(* CODESYS project Bronkhorst.library
   Author: Ziga Javornik
   Version: 0.0.3.1
   Description: Various bronkhorst device impleentations.
   Title: ZigaLibs.Bronkhorst
   Placeholder: ZigaLibs.Bronkhorst
   DefaultNamespace: ZigaLibs.Bronkhorst
   Company: Ziga Javornik

Project tree, tasks and I/O mapping:
  libraries: Tc2_Standard, * (Beckhoff Automation GmbH); Tc2_System, * (Beckhoff Automation GmbH); Tc3_Module, * (Beckhoff Automation GmbH); TcUnit, 1.3.1 (www.tcunit.org); ZigaLibs.Core, 0.0.3.7 (Ziga Javornik); ZigaLibs.Logging, 0.0.4.1 (Ziga Javornik)
  GVLs/
  SOURCE/
    MassFlow or PressureController/
      DUTs/
        data type E_ControllerMode
        data type E_ParameterReadingStep
        data type ST_ControllerCoeList
        data type ST_ControllerInputs
        data type ST_ControllerOutputs
        data type ST_ControllerStatus
      POUs/
        function block FB_FlowController [ST]: FB_init, CalculateMeasuredValue, CalculateSetpointValue, ControllerModeWriting, ControllerSpeedWriting, ReadCoE, Capacity, CapacityUnit, ControllerSpeed, FluidName, Mode, Status
    program FlowUnits [ST]: Bar, LsMin, Sccm, Slm
    program GasTypes [ST]: Air, BBr3, BCl3, C2F6, Cl2, H2, He, N2, O2, SF6, SiF4
  TESTS/
    Test suites/
      function block FB_FlowController_Tests [ST]: Test01_MeasuredValueConversion_1000, Test02_MeasuredValueConversion_32767, Test03_MeasuredValueConversion_0, Test04_MeassuredValueConversion_decimalDigits0, Test05_SetpointValueConversion_1000, Test06_SetpointValueConversion_10000, Test07_SetpointValueConversion_0, Test08_SetpointValueConversion_decimalDigits0, Test09_EnablePreventsOutoutFlowAndSetsControlByteToZero, Test10_ControllerStatusConversion, Test11_ValvePosition
      function block FB_FlowUnits_Tests [ST]: Test_AllFlowUnits
      function block FB_GasTypes_Tests [ST]: Test_AllGasTypes
    program PRG_TESTS [ST]
*)

// SOURCE/MassFlow or PressureController/DUTs/E_ControllerMode
{attribute 'qualified_only'}
{attribute 'to_string'}
TYPE E_ControllerMode :
(
	Controlling 	:= 16#80,	// Control at setpoint value
	ValveClosed		:= 16#83,	// No controller action, valve is closed
	ControllerIdle	:= 16#84,	// No controller action, valve remains its position 
	ValvePurge		:= 16#88	// No controller action, valve is fully open
)USINT;
END_TYPE

// SOURCE/MassFlow or PressureController/DUTs/E_ParameterReadingStep
{attribute 'qualified_only'}
{attribute 'strict'}
TYPE E_ParameterReadingStep :
(
	IDLE,
	GAS_TYPE,
	FLOW_UNIT,
	DECIMAL_DIGITS,
	FLOW_CAPACITY
);
END_TYPE

// SOURCE/MassFlow or PressureController/DUTs/ST_ControllerCoeList
// Contains CoE indexes and sub indexes for Bronkhorst EtherCAT mass flow controller
TYPE ST_ControllerCoeList :
STRUCT
	FluidName		: ZigaLibs_Core.ST_CoeEntry_String30 	:= (Index := 16#2001, SubIndex := 16#12);
	Capacity 		: ZigaLibs_Core.ST_CoeEntry_REAL 		:= (Index := 16#2001, SubIndex := 16#0E);
	CapacityUnit 	: ZigaLibs_Core.ST_CoeEntry_String30 	:= (Index := 16#2001, SubIndex := 16#20);
	DecimalDigits 	: ZigaLibs_Core.ST_CoeEntry_INT 		:= (Index := 16#6407, SubIndex := 16#01);
	ControlMode 	: ZigaLibs_Core.ST_CoeEntry_USINT 		:= (Index := 16#6423, SubIndex := 16#01);
	ControllerSpeed	: ZigaLibs_Core.ST_CoeEntry_USINT		:= (Index := 16#2072, Subindex := 16#1F);
END_STRUCT
END_TYPE

// SOURCE/MassFlow or PressureController/DUTs/ST_ControllerInputs
TYPE ST_ControllerInputs :
STRUCT
	MeassuredValue	: INT;
	ValvePosition	: UINT;
	StatusWord		: UINT;
	AmsAddr			: Tc2_System.ST_AmsAddr;
END_STRUCT
END_TYPE

// SOURCE/MassFlow or PressureController/DUTs/ST_ControllerOutputs
TYPE ST_ControllerOutputs :
STRUCT
	ControlByte	: USINT;
	Setpoint	: INT;
END_STRUCT
END_TYPE

// SOURCE/MassFlow or PressureController/DUTs/ST_ControllerStatus

TYPE ST_ControllerStatus :
STRUCT
	ControllerOn		: BOOL;
	SelfOptimization	: BOOL;
	ManualMode			: BOOL;
	SetpointSwitch		: BOOL;
	OptimizationError	: BOOL;
	DataNotValid		: BOOL;
	Overload			: BOOL;
	NetOverload			: BOOL;
END_STRUCT
END_TYPE

// SOURCE/MassFlow or PressureController/POUs/FB_FlowController
(* Bronkhorst mass flow/pressure controller device implementation.
============================================================================================================================================================================================
CONSTRUCTOR TEMPLATE - COPY EVERYTHING BELOW, ADJUST PARAMETERS ACCORDINGLY!
============================================================================================================================================================================================	
(fPredictedFlowCapacity	:= 100, // [REAL] Predicted flow capacity. If logger is provided and the read capacity differs, the error will be reported by the logger.
sPredictedGasType := N2, // [STRING] Predicted gas type. If logger is provided and the read gas type differs, the error will be reported by the logger.
sPredictedFlowUnit := sccm, // [STRING] Predicted flow unit. If logger is provided and the read flow unit differs, the error will be reported by the logger.
iLogger := 0, // [ZigaLibs_Core.I_LoggerEx] Logger implementation provided, set to 0 if not required.
mode := E_ControllerMode.Controlling); // [E_ControllerMode] Controller initial mode
============================================================================================================================================================================================
*)

FUNCTION_BLOCK FB_FlowController EXTENDS ZigaLibs_Core.FB_HasInstanceNameAndPath
VAR_INPUT
	bEnable				: BOOL;	// Enables controller
	fSetpoint			: REAL;	// Setpoint to the controller
	bReadParameters		: BOOL; // Reads CoE parameters on rising edge trigger
END_VAR
VAR_OUTPUT
	fMeassuredValue	: REAL;	// Measured value, reported from the controller
	fValvePosition	: REAL;	// Valve position
END_VAR

// IO
VAR
	Inputs	AT %I*	: ST_ControllerInputs;
	Outputs	AT %Q* 	: ST_ControllerOutputs;
END_VAR

VAR
	bFirstExecution			: BOOL := TRUE;
	_stringBuilder			: ZigaLibs_Core.FB_StringBuilder;
	_CoeList				: ST_ControllerCoeList;
	_logPrefix				: STRING := Tc2_Standard.CONCAT(STR1 := _instancePath, STR2 := ': ');
	_logger					: REFERENCE TO ZigaLibs_Logging.I_Logger;
	_writeLogs				: BOOL;
	_ethercatBoxName		: Tc2_System.T_MaxString;
	{attribute 'hide'} 
	_mode					: E_ControllerMode;	// Hide since mode switching should be logged (done inside the property setter)
	_status					: ST_ControllerStatus;
	_predictedFlowCapacity	: REAL;
	_predictedGasType		: STRING;
	_predictedFlowUnit		: STRING;
	_writeModeRequired					: BOOL;
	_validateModeWrite					: BOOL;
	_controlModeTmp						: E_ControllerMode;
	_coeReadWrite						: ZigaLibs_Core.FB_CoeReadWrite;
	_readParametersRequest				: Tc2_Standard.R_TRIG;
	_parametersReadingInProgress		: BOOL;
	_readBoxName						: ZigaLibs_Core.FB_ReadBoxName;
	_controllerSpeed					: UINT := 1;
	_updateControllerSpeedRequired		: BOOL;
	_validateControllerSpeed			: BOOL;
END_VAR

VAR CONSTANT
	VALVE_FULLY_OPENED_VALUE : REAL := 617.0;
END_VAR

Outputs.ControlByte := BOOL_TO_BYTE(bEnable);

IF bEnable THEN
	Outputs.Setpoint := CalculateSetpointValue();
ELSE
	Outputs.Setpoint := 0;
END_IF

fMeassuredValue := CalculateMeasuredValue();
fValvePosition := 100.0 * UINT_TO_REAL(Inputs.ValvePosition)/VALVE_FULLY_OPENED_VALUE;

IF bFirstExecution THEN
	IF ReadCoE() THEN
		bFirstExecution := FALSE;
	END_IF
END_IF

_readParametersRequest(CLK := bReadParameters);
// Parameters read request
IF _readParametersRequest.Q THEN
	_parametersReadingInProgress := TRUE;
END_IF

IF _parametersReadingInProgress THEN
	IF ReadCoE() THEN
		_parametersReadingInProgress := FALSE;
	END_IF
END_IF

// Controller mode writing and validation
ControllerModeWriting();
// Controller speed writing and validation
ControllerSpeedWriting();

// Status of the controller
_status.ControllerOn := Inputs.StatusWord.0;
_status.SelfOptimization := Inputs.StatusWord.1;
_status.ManualMode := Inputs.StatusWord.2;
_status.SetpointSwitch := Inputs.StatusWord.3;
_status.OptimizationError := Inputs.StatusWord.4;
_status.DataNotValid := Inputs.StatusWord.8;
_status.Overload := Inputs.StatusWord.9;
_status.NetOverload := Inputs.StatusWord.10;

METHOD FB_init : BOOL
VAR_INPUT
	bInitRetains : BOOL; // if TRUE, the retain variables are initialized (warm start / cold start)
	bInCopyCode : BOOL;  // if TRUE, the instance afterwards gets moved into the copy code (online change)
	
	fPredictedFlowCapacity	: REAL;	// Predicted flow capacity. If bWriteLogs is set to TRUE and the read capacity differs, the error will be reported by the logger.
	sPredictedGasType		: STRING;// Predicted gas type. If bWriteLogs is set to TRUE and the read gas type differs, the error will be reported by the logger.
	sPredictedFlowUnit		: STRING; // Predicted flow unit. If bWriteLogs is set to TRUE and the read flow unit differs, the error will be reported by the logger.
	logger					: REFERENCE TO ZigaLibs_Logging.I_Logger;	// Logger implementation provided, set to 0 if not required.
	mode					: E_ControllerMode;	// Controller initial mode
END_VAR
_predictedFlowCapacity := fPredictedFlowCapacity;
_predictedGasType := sPredictedGasType;
_predictedFlowUnit := sPredictedFlowUnit;
_logger REF= logger;
_mode := mode;
_writeLogs := __ISVALIDREF(logger);
END_METHOD

METHOD PRIVATE CalculateMeasuredValue : REAL
VAR_INPUT
END_VAR
CalculateMeasuredValue :=  INT_TO_REAL(Inputs.MeassuredValue) / LREAL_TO_REAL(EXPT(10,_CoeList.DecimalDigits.Value));
END_METHOD

METHOD PRIVATE CalculateSetpointValue : INT
VAR_INPUT
END_VAR
CalculateSetpointValue := REAL_TO_INT(fSetpoint * LREAL_TO_REAL(EXPT(10, _CoeList.DecimalDigits.Value)));
END_METHOD

METHOD PRIVATE ControllerModeWriting
IF _writeModeRequired AND_THEN _coeReadWrite.WriteAny(
		CoeEntry := ADR(_CoeList.ControlMode),
		Value := _mode,
		SlaveAddr := Inputs.AmsAddr)
THEN
	IF _writeLogs THEN
		_logger.LogInfo(message := _stringBuilder.Reset()
			.AddString(str := _logPrefix)
			.AddString(str := 'Finished writing control mode for EtherCAT device ')
			.AddWithDblQuotationMarks(str := _ethercatBoxName)
			.AddString(str := '.')
			.Create());
	END_IF
	_validateModeWrite := TRUE;
	_writeModeRequired := FALSE;
END_IF

IF _validateModeWrite AND_THEN _coeReadWrite.ReadAny(
		CoeEntry := ADR(_CoeList.ControlMode),
		Value := _CoeList.ControlMode.Value,
		SlaveAddr := Inputs.AmsAddr)
THEN
	_validateModeWrite := FALSE;
	IF _writeLogs THEN
		IF _CoeList.ControlMode.Value <> _mode THEN
			// This allows for using TO_STRING on the enum value for better logging experience.
			_controlModeTmp := _CoeList.ControlMode.Value;
			_logger.LogError(message := _stringBuilder.Reset()
				.AddString(str := _logPRefix)
				.AddString('Control mode validation failed! Actual mode read is ')
				.AddWithDblQuotationMarks(str := TO_STRING(_controlModeTmp))
				.AddString(' required mode is ')
				.AddWithDblQuotationMarks(str := TO_STRING(_mode))
				.Create());
		ELSE
			_logger.LogInfo(message := _stringBuilder.Reset()
				.AddString(str := _logPrefix)
				.AddString('Control mode setting validation successful.')
				.Create());
		END_IF
	END_IF
END_IF
END_METHOD

METHOD PRIVATE ControllerSpeedWriting
VAR_INPUT
END_VAR
IF _updateControllerSpeedRequired AND_THEN _coeReadWrite.WriteAny(
		CoeEntry := ADR(_CoeList.ControllerSpeed),
		Value := _controllerSpeed,
		SlaveAddr := Inputs.AmsAddr)
THEN
	IF _writeLogs THEN
	_logger.LogInfo(message := _stringBuilder.Reset()
		.AddString(str := _logPrefix)
		.AddString(str := 'Finished writing controller speed for EtherCAT device ')
		.AddWithDblQuotationMarks(str := _ethercatBoxName)
		.AddString(str := '.')
		.Create());
	END_IF
	_validateControllerSpeed := TRUE;
	_updateControllerSpeedRequired := FALSE;
END_IF

IF _validateControllerSpeed AND_THEN _coeReadWrite.ReadAny(
		CoeEntry := ADR(_CoeList.ControllerSpeed),
		Value := _CoeList.ControlMode.Value,
		SlaveAddr := Inputs.AmsAddr)
THEN
	_validateControllerSpeed := FALSE;
	IF _writeLogs THEN
		IF _CoeList.ControlMode.Value <> _mode THEN
			_logger.LogError(message := _stringBuilder.Reset()
				.AddString(str := _logPRefix)
				.AddString('Control speed validation failed! Actual speed read is ')
				.AddWithDblQuotationMarks(str := TO_STRING(_CoeList.ControllerSpeed.Value))
				.AddString(' required speed is ')
				.AddWithDblQuotationMarks(str := TO_STRING(_controllerSpeed))
				.Create());
		ELSE
			_logger.LogInfo(message := _stringBuilder.Reset()
				.AddString(str := _logPrefix)
				.AddString('Control speed setting validation successful.')
				.Create());
		END_IF
	END_IF
END_IF
END_METHOD

(* Reads CoE items and updates them. Returns TRUE when done, even if an error occurs. Error is reported to log.*)
METHOD PRIVATE ReadCoE : BOOL
VAR_INST
	eReadCoeStep	: E_ParameterReadingStep;
	bCoeReadError	: BOOL;
	bError			: BOOL;
	fbCoeReadWrite	: ZigaLibs_Core.FB_CoeReadWrite;
END_VAR

VAR CONSTANT
	MAX_REAL_VALUE_DEVIATION : REAL := 0.1;
END_VAR

VAR_INST
	message	: Tc2_System.T_MaxString;
	mfcName	: Tc2_System.T_MaxString;
END_VAR
CASE eReadCoeStep OF
	E_ParameterReadingStep.IDLE:
		ReadCoE := FALSE;
		message := '';
		IF _ethercatBoxName = '' THEN
			_readBoxName(
				AmsNetId := Inputs.AmsAddr,
				PlcRuntimeNetId := '',
				error => bError,
				name => _ethercatBoxName);
		ELSIF _ethercatBoxName <> '' OR bError THEN
			eReadCoeStep := E_ParameterReadingStep.GAS_TYPE;
			IF _writeLogs THEN
				IF NOT bError THEN
					message := _stringBuilder.Reset()	
						.AddString(str := _logPrefix)
						.AddString(str := 'MFC parameters ')
						.AddWithDblQuotationMarks(str := _ethercatBoxName)
						.AddString(str := ':')
						.Create();
				ELSE
					_logger.LogInfo(message := _stringBuilder.Reset()	
						.AddString(str := _logPrefix)
						.AddString(str := 'Reading CoE parameters for Bronkhorst device ')
						.AddWithDblQuotationMarks(str := '<Error reading EC box name>')
						.AddString(str := '...')
						.Create());
				END_IF

			END_IF
		END_IF
		
	E_ParameterReadingStep.GAS_TYPE:
		IF fbCoeReadWrite.ReadAny(
			CoeEntry := ADR(_CoeList.FluidName),
			Value := _CoeList.FluidName.Value,
			SlaveAddr := Inputs.AmsAddr)
		THEN
			_CoeList.FluidName.Value := ZigaLibs_Core.StringHelper.TrimRightSide(_CoeList.FluidName.Value);
			IF _writeLogs THEN
				IF ZigaLibs_Core.StringHelper.TrimRightSide(_CoeList.FluidName.Value) <> _predictedGasType THEN
					_logger.LogWarning(message := _stringBuilder.Reset()
						.AddString(_logPrefix)
						.AddString('Invalid gas type found! Predicted gas type is ')
						.AddWithDblQuotationMarks(_predictedGasType)
						.AddString(' and actual gas type found is ')
						.AddWithDblQuotationMarks(_coeList.FluidName.Value)
						.Create());
				ELSE
					message :=_stringBuilder.Reset()
						.AddString(message)
						.AddString('[')
						.AddString('Gas type: ')
						.AddWithDblQuotationMarks(_coeList.FluidName.Value)
						.AddString(']')
						.Create();
				END_IF
			END_IF
			eReadCoeStep := E_ParameterReadingStep.FLOW_UNIT;
		END_IF
		
	E_ParameterReadingStep.FLOW_UNIT:
		IF fbCoeReadWrite.ReadAny(
			CoeEntry := ADR(_CoeList.CapacityUnit),
			Value := _CoeList.CapacityUnit.Value,
			SlaveAddr := Inputs.AmsAddr)
		THEN
			_CoeList.CapacityUnit.Value := ZigaLibs_Core.StringHelper.TrimRightSide(_CoeList.CapacityUnit.Value);
			IF _writeLogs THEN
				IF ZigaLibs_Core.StringHelper.TrimRightSide(_CoeList.CapacityUnit.Value) <> _predictedFlowUnit THEN
					_logger.LogWarning(message := _stringBuilder.Reset()
						.AddString(_logPrefix)
						.AddString('Invalid flow unit found! Predicted unit is ')
						.AddWithDblQuotationMarks(_predictedFlowUnit)
						.AddString(' and actual flow unit found is ')
						.AddWithDblQuotationMarks(_coeList.CapacityUnit.Value)
						.Create());				
				ELSE
					message :=_stringBuilder.Reset()
						.AddString(message)
						.AddString('[')
						.AddString('Flow unit: ')
						.AddWithDblQuotationMarks(_coeList.CapacityUnit.Value)
						.AddString(']')
						.Create();
				END_IF
			END_IF
			eReadCoeStep := E_ParameterReadingStep.DECIMAL_DIGITS;
		END_IF
		
	E_ParameterReadingStep.DECIMAL_DIGITS:
		IF fbCoeReadWrite.ReadAny(
			CoeEntry := ADR(_CoeList.DecimalDigits),
			Value := _CoeList.DecimalDigits.Value,
			SlaveAddr := Inputs.AmsAddr)
		THEN
			eReadCoeStep := E_ParameterReadingStep.FLOW_CAPACITY;
		END_IF
		
	E_ParameterReadingStep.FLOW_CAPACITY:
		IF fbCoeReadWrite.ReadAny(
			CoeEntry := ADR(_CoeList.Capacity),
			Value := _CoeList.Capacity.Value,
			SlaveAddr := Inputs.AmsAddr)
		THEN
			IF _writeLogs THEN
				IF ABS(_CoeList.Capacity.Value - _predictedFlowCapacity) >= MAX_REAL_VALUE_DEVIATION THEN
					_logger.LogWarning(message := _stringBuilder.Reset()
						.AddString(_logPrefix)
						.AddString('Invalid flow capacity found! Predicted capacity is ')
						.AddString(ZigaLibs_Core.StringConstants.DoubleQuotationMark)
						.AddAnyReal(_predictedFlowCapacity, 3, TRUE).AddString(' ').AddString(_coeList.CapacityUnit.Value)
						.AddString(ZigaLibs_Core.StringConstants.DoubleQuotationMark)
						.AddString(' and actual flow capacity found is ')
						.AddString(ZigaLibs_Core.StringConstants.DoubleQuotationMark)
						.AddAnyReal(_CoeList.Capacity.Value, 3, TRUE).AddString(' ').AddString(_coeList.CapacityUnit.Value)
						.AddString(ZigaLibs_Core.StringConstants.DoubleQuotationMark)
						.AddString('!')
						.Create());
					ELSE
							
					message :=_stringBuilder.Reset()
						.AddString(message)
						.AddString('[')
						.AddString('Flow capacity: ')
						.AddString(ZigaLibs_Core.StringConstants.DoubleQuotationMark)
						.AddAnyReal(_CoeList.Capacity.Value, 3, TRUE).AddString(' ').AddString(_coeList.CapacityUnit.Value)
						.AddString(ZigaLibs_Core.StringConstants.DoubleQuotationMark)
						.AddString(']')
						.Create();
						
					_logger.LogInfo(message);
					END_IF
				END_IF
			eReadCoeStep := E_ParameterReadingStep.IDLE;
			ReadCoE := TRUE;
		END_IF	
END_CASE
END_METHOD

{attribute 'monitoring':='call'}
// Gets capacity of the device
PROPERTY Capacity : REAL
GET
Capacity := _CoeList.Capacity.Value;
END_GET
END_PROPERTY

{attribute 'monitoring':='call'}
// Gets the capacity unit of the device
PROPERTY CapacityUnit : STRING(30)
GET
CapacityUnit := _CoeList.CapacityUnit.Value;
END_GET
END_PROPERTY

{attribute 'monitoring'='call'}
(*Gets or sets the controller speed.
The controller speed is default set on 1, increasing THIS number will make it faster. 
Please be aware that increasing the controller speed can lead to oscillation when setpoint steps are to steep, 
this will need to be fine-tuned on site to find the optimum setting for the process*)
PROPERTY PUBLIC ControllerSpeed : UINT := 1
GET
ControllerSpeed := _controllerSpeed;
END_GET
SET
IF ControllerSpeed <> _controllerSpeed THEN
	_updateControllerSpeedRequired := TRUE;
END_IF
_controllerSpeed := ControllerSpeed;
END_SET
END_PROPERTY

{attribute 'monitoring':='call'}
// Gets the fluid name of the device
PROPERTY FluidName : STRING(30)
GET
FluidName := _CoeList.FluidName.Value;
END_GET
END_PROPERTY

{attribute 'monitoring':='call'}
// Gets or sets the controller mode
PROPERTY PUBLIC Mode : E_ControllerMode
GET
Mode := _mode;
END_GET
SET
IF _mode <> Mode THEN
	_writeModeRequired := TRUE;
END_IF

_mode := Mode;
END_SET
END_PROPERTY

{attribute 'monitoring':='call'}
// Gets the controller status
PROPERTY Status : REFERENCE TO ST_ControllerStatus
GET
Status REF= _status;
END_GET
END_PROPERTY

END_FUNCTION_BLOCK

// SOURCE/FlowUnits
PROGRAM FlowUnits
VAR
END_VAR

PROPERTY Bar : string
GET
Bar := 'bar(g)';
END_GET
END_PROPERTY

PROPERTY PUBLIC LsMin : STRING
GET
LsMin := 'ls/min';
END_GET
END_PROPERTY

PROPERTY Sccm : STRING
GET
Sccm := 'sccm';
END_GET
END_PROPERTY

PROPERTY Slm : STRING
GET
Slm := 'slm';
END_GET
END_PROPERTY

END_PROGRAM

// SOURCE/GasTypes
{attribute 'no_explicit_call' := 'Body contains no logic, calling methods only allowed.'}
{attribute 'hide_all_locals'}

// A class containing possible gas types for Bronkhorst devices stored as a string.
PROGRAM GasTypes
VAR
END_VAR

{attribute 'monitoring':='call}
PROPERTY Air : STRING
GET
Air := 'AiR';
END_GET
END_PROPERTY

{attribute 'monitoring':='variable'}
PROPERTY BBr3 : STRING
GET
BBr3 := 'BBr3';
END_GET
END_PROPERTY

{attribute 'monitoring':='variable'}
PROPERTY BCl3 : STRING
GET
BCl3 := 'BCl3';
END_GET
END_PROPERTY

{attribute 'monitoring':='variable'}
PROPERTY C2F6 : STRING
GET
C2F6 := 'C2F6';
END_GET
END_PROPERTY

{attribute 'monitoring':='variable'}
PROPERTY Cl2 : STRING
GET
Cl2 := 'Cl2';
END_GET
END_PROPERTY

{attribute 'monitoring':='variable'}
PROPERTY H2 : STRING
GET
H2 := 'H2';
END_GET
END_PROPERTY

{attribute 'monitoring':='variable'}
PROPERTY He : STRING
GET
He := 'He';
END_GET
END_PROPERTY

{attribute 'monitoring':='variable'}
PROPERTY N2 : STRING
GET
N2 := 'N2';
END_GET
END_PROPERTY

{attribute 'monitoring':='variable'}
PROPERTY O2 : STRING
GET
O2 := 'O2';
END_GET
END_PROPERTY

{attribute 'monitoring':='variable'}
PROPERTY SF6 : STRING
GET
SF6 := 'SF6';
END_GET
END_PROPERTY

{attribute 'monitoring':='variable'}
PROPERTY SiF4 : STRING
GET
SiF4 := 'SiF4';
END_GET
END_PROPERTY

END_PROGRAM

// TESTS/Test suites/FB_FlowController_Tests
// Subject under test
FUNCTION_BLOCK INTERNAL FB_FlowController_Tests EXTENDS TcUnit.FB_TestSuite

// Create instance variables that will be accesible for all tests
VAR
	_mfc : FB_FlowController(	
		fPredictedFlowCapacity	:= 0.0,	// Predicted flow capacity. If bLogInvalidParams is set to TRUE and the read capacity differs, the error will be reported by the logger.
		sPredictedGasType		:= 'Cl2',// Predicted gas type. If bLogInvalidParams is set to TRUE and the read gas type differs, the error will be reported by the logger.
		sPredictedFlowUnit		:= 'sccm', // Predicted flow unit. If bLogInvalidParams is set to TRUE and the read flow unit differs, the error will be reported by the logger.
		logger					:= 0,	// Logger implementation provided
		mode					:= E_ControllerMode.Controlling);
END_VAR

// Call your test methods here
Test01_MeasuredValueConversion_1000();
Test02_MeasuredValueConversion_32767();
Test03_MeasuredValueConversion_0();
Test04_MeassuredValueConversion_decimalDigits0();
Test05_SetpointValueConversion_1000();
Test06_SetpointValueConversion_10000();
Test07_SetpointValueConversion_0();
Test08_SetpointValueConversion_decimalDigits0();
Test09_EnablePreventsOutoutFlowAndSetsControlByteToZero();
Test10_ControllerStatusConversion();
Test11_ValvePosition();

METHOD PRIVATE Test01_MeasuredValueConversion_1000

(* Instanced variables are VERY useful for writing tests since tests are run in paralel (by default).
By instantiating local variables that are not placed on the same stack as method (values are retained between calls)
you make sure that the SUT is not changed by some other test. *)

// Place temporary variables here
VAR
	
END_VAR
// The name of the test, is the same as method name!
IF TcUnit.TEST_ORDERED('Test01_MeasuredValueConversion_1000') THEN

	TcUnit.WRITE_PROTECTED_INT(
		Ptr := ADR(_mfc.Inputs),
		Value := 1000);
		
	TcUnit.WRITE_PROTECTED_INT(
		Ptr := ADR(_mfc._coeList.DecimalDigits.Value),
		Value := 2);
		
	_mfc();	
	
	AssertEquals_REAL(
		Actual := _mfc.fMeassuredValue,
		Expected := 1000.0 / EXPT(10,2),
		Delta := 0.1,
		Message := 'Masured flow is calculated incorectly!');
		
	TcUnit.TEST_FINISHED();
END_IF
END_METHOD

METHOD PRIVATE Test02_MeasuredValueConversion_32767

(* Instanced variables are VERY useful for writing tests since tests are run in paralel (by default).
By instantiating local variables that are not placed on the same stack as method (values are retained between calls)
you make sure that the SUT is not changed by some other test. *)
VAR_INST

END_VAR

// Place temporary variables here
VAR
	
END_VAR
// The name of the test, is the same as method name!
IF TcUnit.TEST_ORDERED('Test02_MeasuredValueConversion_32767') THEN

	TcUnit.WRITE_PROTECTED_INT(
		Ptr := ADR(_mfc.Inputs),
		Value := 32767);
		
	TcUnit.WRITE_PROTECTED_INT(
		Ptr := ADR(_mfc._coeList.DecimalDigits.Value),
		Value := 2);
		
	_mfc();	
	
	AssertEquals_REAL(
		Actual := _mfc.fMeassuredValue,
		Expected := 32767.0 / EXPT(10,2),
		Delta := 0.1,
		Message := 'Masured flow is calculated incorectly!');
		
	TcUnit.TEST_FINISHED();
END_IF
END_METHOD

METHOD PRIVATE Test03_MeasuredValueConversion_0

(* Instanced variables are VERY useful for writing tests since tests are run in paralel (by default).
By instantiating local variables that are not placed on the same stack as method (values are retained between calls)
you make sure that the SUT is not changed by some other test. *)

// Place temporary variables here
VAR
	
END_VAR
// The name of the test, is the same as method name!
IF TcUnit.TEST_ORDERED('Test03_MeasuredValueConversion_0') THEN

	TcUnit.WRITE_PROTECTED_INT(
		Ptr := ADR(_mfc.Inputs),
		Value := 0);
		
	TcUnit.WRITE_PROTECTED_INT(
		Ptr := ADR(_mfc._coeList.DecimalDigits.Value),
		Value := 2);
		
	_mfc();	
	
	AssertEquals_REAL(
		Actual := _mfc.fMeassuredValue,
		Expected := 0,
		Delta := 0.1,
		Message := 'Masured flow is calculated incorectly!');
		
	TcUnit.TEST_FINISHED();
END_IF
END_METHOD

METHOD PRIVATE Test04_MeassuredValueConversion_decimalDigits0

(* Instanced variables are VERY useful for writing tests since tests are run in paralel (by default).
By instantiating local variables that are not placed on the same stack as method (values are retained between calls)
you make sure that the SUT is not changed by some other test. *)
VAR_INST
END_VAR

// Place temporary variables here
VAR
	
END_VAR
// The name of the test, is the same as method name!
IF TcUnit.TEST_ORDERED('Test04_MeassuredValueConversion_decimalDigits0') THEN

	TcUnit.WRITE_PROTECTED_INT(
		Ptr := ADR(_mfc.Inputs),
		Value := 30000);
		
	TcUnit.WRITE_PROTECTED_INT(
		Ptr := ADR(_mfc._coeList.DecimalDigits.Value),
		Value := 0);
		
	_mfc();	
	
	AssertEquals_REAL(
		Actual := _mfc.fMeassuredValue,
		Expected := 30000,
		Delta := 0.1,
		Message := 'Masured flow with decimal digits value being 0 is calculated incorectly!');
		
	TcUnit.TEST_FINISHED();
END_IF
END_METHOD

METHOD PRIVATE Test05_SetpointValueConversion_1000

(* Instanced variables are VERY useful for writing tests since tests are run in paralel (by default).
By instantiating local variables that are not placed on the same stack as method (values are retained between calls)
you make sure that the SUT is not changed by some other test. *)

// Place temporary variables here
VAR
	
END_VAR
// The name of the test, is the same as method name!
IF TcUnit.TEST_ORDERED('Test05_SetpointValueConversion_1000') THEN

	TcUnit.WRITE_PROTECTED_INT(
		Ptr := ADR(_mfc._coeList.DecimalDigits.Value),
		Value := 1);
		
	_mfc(bEnable := TRUE, fSetpoint := 1000);	
	
	AssertEquals_REAL(
		Actual := _mfc.Outputs.Setpoint,
		Expected := 1000.0 * EXPT(10,1),
		Delta := 0.1,
		Message := 'Setpoint flow is calculated incorectly!');
		
	TcUnit.TEST_FINISHED();
END_IF
END_METHOD

METHOD PRIVATE Test06_SetpointValueConversion_10000

(* Instanced variables are VERY useful for writing tests since tests are run in paralel (by default).
By instantiating local variables that are not placed on the same stack as method (values are retained between calls)
you make sure that the SUT is not changed by some other test. *)
VAR_INST
	
END_VAR

// Place temporary variables here
VAR
	
END_VAR
// The name of the test, is the same as method name!
IF TcUnit.TEST_ORDERED('Test06_SetpointValueConversion_10000') THEN
	TcUnit.WRITE_PROTECTED_INT(
		Ptr := ADR(_mfc._coeList.DecimalDigits.Value),
		Value := 0);
		
	_mfc(bEnable := TRUE, fSetpoint := 10_000.0);	
	
	AssertEquals_REAL(
		Actual := _mfc.Outputs.Setpoint,
		Expected := 10_000.0,
		Delta := 0.1,
		Message := 'Setpoint flow is calculated incorectly!');
		
	TcUnit.TEST_FINISHED();
END_IF
END_METHOD

METHOD PRIVATE Test07_SetpointValueConversion_0

(* Instanced variables are VERY useful for writing tests since tests are run in paralel (by default).
By instantiating local variables that are not placed on the same stack as method (values are retained between calls)
you make sure that the SUT is not changed by some other test. *)

// Place temporary variables here
VAR
	
END_VAR
// The name of the test, is the same as method name!
IF TcUnit.TEST_ORDERED('Test07_SetpointValueConversion_0') THEN
	
		
	TcUnit.WRITE_PROTECTED_INT(
		Ptr := ADR(_mfc._coeList.DecimalDigits.Value),
		Value := 3);
		
	_mfc(bEnable := TRUE, fSetpoint := 0.0);	
	
	AssertEquals_REAL(
		Actual := _mfc.Outputs.Setpoint,
		Expected := 0,
		Delta := 0.1,
		Message := 'Setpoint flow is calculated incorectly!');
		
	TcUnit.TEST_FINISHED();
END_IF
END_METHOD

METHOD PRIVATE Test08_SetpointValueConversion_decimalDigits0

(* Instanced variables are VERY useful for writing tests since tests are run in paralel (by default).
By instantiating local variables that are not placed on the same stack as method (values are retained between calls)
you make sure that the SUT is not changed by some other test. *)
VAR_INST
END_VAR

// Place temporary variables here
VAR
	
END_VAR
// The name of the test, is the same as method name!
IF TcUnit.TEST_ORDERED('Test08_SetpointValueConversion_decimalDigits0') THEN
	
	TcUnit.WRITE_PROTECTED_INT(
		Ptr := ADR(_mfc._coeList.DecimalDigits.Value),
		Value := 0);
		
	_mfc(bEnable := TRUE, fSetpoint := 30_000.0);	
	
	AssertEquals_REAL(
		Actual := _mfc.Outputs.Setpoint,
		Expected := 30000,
		Delta := 0.1,
		Message := 'Masured flow with decimal digits value being 0 is calculated incorectly!');
		
	TcUnit.TEST_FINISHED();
END_IF
END_METHOD

METHOD Test09_EnablePreventsOutoutFlowAndSetsControlByteToZero
VAR_INPUT
END_VAR
IF TcUnit.TEST_ORDERED('Test09_EnablePreventsOutoutFlowAndSetsControlByteToZero') THEN

	TcUnit.WRITE_PROTECTED_INT(
		Ptr := ADR(_mfc._coeList.DecimalDigits.Value),
		Value := 0);
		
	_mfc(bEnable := TRUE, fSetpoint := 10_000.0);
	AssertEquals_REAL(
		Actual := _mfc.Outputs.Setpoint,
		Expected := 10_000.0,
		Delta := 0.1,
		Message := 'When controller is enabled, flow should be set to the output!');
		
	AssertEquals_BYTE(
		Actual := _mfc.Outputs.ControlByte,
		Expected := 1,
		Message := 'If controller is enabled, control byte value should be 1');
		
	_mfc(bEnable := FALSE, fSetpoint := 10_000.0);
	AssertEquals_REAL(
		Actual := _mfc.Outputs.Setpoint,
		Expected := 0.0,
		Delta := 0.1,
		Message := 'When controller is disabled, flow should be set to zero!');
		
	AssertEquals_BYTE(
		Actual := _mfc.Outputs.ControlByte,
		Expected :=0,
		Message := 'If controller is disabled, control byte value should be 0');
	
	TcUnit.TEST_FINISHED();
END_IF
END_METHOD

METHOD Test10_ControllerStatusConversion
VAR_INPUT
END_VAR
VAR_INST
	statusWord	: WORD;
END_VAR
IF TcUnit.TEST_ORDERED('Test10_ControllerStatusConversion') THEN
	TcUnit.WRITE_PROTECTED_WORD(
		Ptr := ADR(_mfc.Inputs.StatusWord),
		Value := statusWord);
		
	_mfc();
	AssertTrue(
		Condition := _mfc.Status.ControllerOn = FALSE AND
					_mfc.Status.DataNotValid = FALSE AND
					_mfc.Status.ManualMode = FALSE AND
					_mfc.Status.NetOverload = FALSE AND
					_mfc.Status.OptimizationError = FALSE AND
					_mfc.Status.Overload = FALSE AND
					_mfc.Status.SelfOptimization = FALSE AND
					_mfc.Status.SetpointSwitch = FALSE,
		Message := 'Incorrect status conversion for all status false!');	
		
	statusWord.0 := TRUE;	
	TcUnit.WRITE_PROTECTED_WORD(
		Ptr := ADR(_mfc.Inputs.StatusWord),
		Value := statusWord);
	
	_mfc();
	AssertTrue(
		Condition := _mfc.Status.ControllerOn = TRUE AND
					_mfc.Status.SelfOptimization = FALSE AND
					_mfc.Status.ManualMode = FALSE AND
					_mfc.Status.SetpointSwitch = FALSE AND
					_mfc.Status.OptimizationError = FALSE AND
					_mfc.Status.DataNotValid = FALSE AND
					_mfc.Status.Overload = FALSE AND
					_mfc.Status.NetOverload = FALSE,
		Message := 'Incorrect status conversion for Controller On!');	
		
	statusWord.1 := TRUE;		
	TcUnit.WRITE_PROTECTED_WORD(
		Ptr := ADR(_mfc.Inputs.StatusWord),
		Value := statusWord);
	
	_mfc();
	AssertTrue(
		Condition := _mfc.Status.ControllerOn = TRUE AND
					_mfc.Status.SelfOptimization = TRUE AND
					_mfc.Status.ManualMode = FALSE AND
					_mfc.Status.SetpointSwitch = FALSE AND
					_mfc.Status.OptimizationError = FALSE AND
					_mfc.Status.DataNotValid = FALSE AND
					_mfc.Status.Overload = FALSE AND
					_mfc.Status.NetOverload = FALSE,
		Message := 'Incorrect status conversion SelfOptimization!');	
	
	statusWord.2 := TRUE;		
	TcUnit.WRITE_PROTECTED_WORD(
		Ptr := ADR(_mfc.Inputs.StatusWord),
		Value := statusWord);
	
	_mfc();
	AssertTrue(
		Condition := _mfc.Status.ControllerOn = TRUE AND
					_mfc.Status.SelfOptimization = TRUE AND
					_mfc.Status.ManualMode = TRUE AND
					_mfc.Status.SetpointSwitch = FALSE AND
					_mfc.Status.OptimizationError = FALSE AND
					_mfc.Status.DataNotValid = FALSE AND
					_mfc.Status.Overload = FALSE AND
					_mfc.Status.NetOverload = FALSE,
		Message := 'Incorrect status conversion ManualMode!');	
	
	statusWord.3 := TRUE;		
	TcUnit.WRITE_PROTECTED_WORD(
		Ptr := ADR(_mfc.Inputs.StatusWord),
		Value := statusWord);
	
	_mfc();
	AssertTrue(
		Condition := _mfc.Status.ControllerOn = TRUE AND
					_mfc.Status.SelfOptimization = TRUE AND
					_mfc.Status.ManualMode = TRUE AND
					_mfc.Status.SetpointSwitch = TRUE AND
					_mfc.Status.OptimizationError = FALSE AND
					_mfc.Status.DataNotValid = FALSE AND
					_mfc.Status.Overload = FALSE AND
					_mfc.Status.NetOverload = FALSE,
		Message := 'Incorrect status conversion for SetpointSwitch!');	
	
	statusWord.4 := TRUE;
	TcUnit.WRITE_PROTECTED_WORD(
		Ptr := ADR(_mfc.Inputs.StatusWord),
		Value := statusWord);
	
	_mfc();
	AssertTrue(
		Condition := _mfc.Status.ControllerOn = TRUE AND
					_mfc.Status.SelfOptimization = TRUE AND
					_mfc.Status.ManualMode = TRUE AND
					_mfc.Status.SetpointSwitch = TRUE AND
					_mfc.Status.OptimizationError = TRUE AND
					_mfc.Status.DataNotValid = FALSE AND
					_mfc.Status.Overload = FALSE AND
					_mfc.Status.NetOverload = FALSE,
		Message := 'Incorrect status conversion OptimizationError!');	
	
	statusWord.8 := TRUE;	
	TcUnit.WRITE_PROTECTED_WORD(
		Ptr := ADR(_mfc.Inputs.StatusWord),
		Value := statusWord);
	
	_mfc();
	AssertTrue(
		Condition := _mfc.Status.ControllerOn = TRUE AND
					_mfc.Status.SelfOptimization = TRUE AND
					_mfc.Status.ManualMode = TRUE AND
					_mfc.Status.SetpointSwitch = TRUE AND
					_mfc.Status.OptimizationError = TRUE AND
					_mfc.Status.DataNotValid = TRUE AND
					_mfc.Status.Overload = FALSE AND
					_mfc.Status.NetOverload = FALSE,
		Message := 'Incorrect status conversion for DataNotValid!');	
	
	statusWord.9 := TRUE;		
	TcUnit.WRITE_PROTECTED_WORD(
		Ptr := ADR(_mfc.Inputs.StatusWord),
		Value := statusWord);
	
	_mfc();
	AssertTrue(
		Condition := _mfc.Status.ControllerOn = TRUE AND
					_mfc.Status.SelfOptimization = TRUE AND
					_mfc.Status.ManualMode = TRUE AND
					_mfc.Status.SetpointSwitch = TRUE AND
					_mfc.Status.OptimizationError = TRUE AND
					_mfc.Status.DataNotValid = TRUE AND
					_mfc.Status.Overload = TRUE AND
					_mfc.Status.NetOverload = FALSE,
		Message := 'Incorrect status conversion for Overload!');	
	
	statusWord.10 := TRUE;
	TcUnit.WRITE_PROTECTED_WORD(
		Ptr := ADR(_mfc.Inputs.StatusWord),
		Value := statusWord);
	
	_mfc();
	AssertTrue(
		Condition := _mfc.Status.ControllerOn = TRUE AND
					_mfc.Status.SelfOptimization = TRUE AND
					_mfc.Status.ManualMode = TRUE AND
					_mfc.Status.SetpointSwitch = TRUE AND
					_mfc.Status.OptimizationError = TRUE AND
					_mfc.Status.DataNotValid = TRUE AND
					_mfc.Status.Overload = TRUE AND
					_mfc.Status.NetOverload = TRUE,
		Message := 'Incorrect status conversion for NetOverload!');	
	
	TcUnit.TEST_FINISHED();
END_IF
END_METHOD

METHOD Test11_ValvePosition
VAR_INPUT
END_VAR


VAR CONSTANT
	VALVE_FULLY_OPENED_VALUE	: UINT := 617;
END_VAR
IF TcUnit.TEST_ORDERED('Test11_ValvePosition') THEN
	
	// Fully closed
	TcUnit.WRITE_PROTECTED_UINT(
		Ptr := ADR(_mfc.Inputs.ValvePosition), 
		Value := 0);
		
	_mfc();
	AssertEquals_REAL(
		Expected := 0,
		Actual := _mfc.fValvePosition,
		Delta := 0.1,
		Message := 'When valve position is 0, expected output should be 0');

	// Half opened	
	TcUnit.WRITE_PROTECTED_UINT(
		Ptr :=	ADR(_mfc.Inputs.ValvePosition), 
		Value := VALVE_FULLY_OPENED_VALUE/2);
		
	_mfc();
	AssertEquals_REAL(
		Expected := 49.9,
		Actual := _mfc.fValvePosition,
		Delta := 0.2,
		Message := 'When valve position is 308, expected output should be 49.9');
	
	// Fully opened
	TcUnit.WRITE_PROTECTED_UINT(
		Ptr := ADR(_mfc.Inputs.ValvePosition), 
		Value := VALVE_FULLY_OPENED_VALUE);
		
	_mfc();	
	AssertEquals_REAL(
		Expected := 100,
		Actual := _mfc.fValvePosition,
		Delta := 0.1,
		Message := 'When valve position is 617, expected output should be 100');		
		
	TcUnit.TEST_FINISHED();
END_IF
END_METHOD

END_FUNCTION_BLOCK

// TESTS/Test suites/FB_FlowUnits_Tests
FUNCTION_BLOCK FB_FlowUnits_Tests EXTENDS TcUnit.FB_TestSuite
VAR_INPUT
END_VAR
VAR_OUTPUT
END_VAR
VAR
END_VAR

Test_AllFlowUnits();

METHOD Test_AllFlowUnits
VAR_INPUT
END_VAR
TcUnit.TEST('Test_AllFlowUnits');

AssertEquals_STRING('slm', FlowUnits.Slm, 'Returned property value is incorrect.');
AssertEquals_STRING('sccm', FlowUnits.Sccm, 'Returned property value is incorrect.');
AssertEquals_STRING('bar(g)', FlowUnits.Bar, 'Returned property value is incorrect.');

TcUnit.TEST_FINISHED();
END_METHOD

END_FUNCTION_BLOCK

// TESTS/Test suites/FB_GasTypes_Tests
FUNCTION_BLOCK FB_GasTypes_Tests EXTENDS TcUnit.FB_TestSuite
VAR_INPUT
END_VAR
VAR_OUTPUT
END_VAR
VAR
END_VAR

Test_AllGasTypes();

METHOD Test_AllGasTypes
VAR_INPUT
END_VAR
TcUnit.TEST('Test_AllGasTypes');

AssertEquals_STRING('BBr3', GasTypes.BBr3, 'Returned property value is incorrect.');
AssertEquals_STRING('BCl3', GasTypes.BCl3, 'Returned property value is incorrect.');
AssertEquals_STRING('Cl2', GasTypes.Cl2, 'Returned property value is incorrect.');
AssertEquals_STRING('H2', GasTypes.H2, 'Returned property value is incorrect.');
AssertEquals_STRING('He', GasTypes.He, 'Returned property value is incorrect.');
AssertEquals_STRING('N2', GasTypes.N2, 'Returned property value is incorrect.');
AssertEquals_STRING('O2', GasTypes.O2, 'Returned property value is incorrect.');
AssertEquals_STRING('SF6', GasTypes.SF6, 'Returned property value is incorrect.');
AssertEquals_STRING('SiF4', GasTypes.SiF4, 'Returned property value is incorrect.');

TcUnit.TEST_FINISHED();
END_METHOD

END_FUNCTION_BLOCK

// TESTS/PRG_TESTS
PROGRAM INTERNAL PRG_TESTS

(* Instantiate test suites here. Naming convention for tests should be a suffix with _Tests.
Good practice for creating test methods is to end them with _test as well. *)
VAR
	FlowControllerTests	: FB_FlowController_Tests;
	FlowUnitTests		: FB_FlowUnits_Tests;
	GasTypesTests		: FB_GasTypes_Tests;
END_VAR

// Run tests in paralel
//TcUnit.RUN();

// Run tests in sequence, one after the other. Uncomment if required.
TcUnit.RUN_IN_SEQUENCE();

END_PROGRAM
